# EPICS substitutions: db/ecmcEL37X2_50.substitutions
file ecmcEL37XX-chX.template
{
  pattern { CH_ID, DTYP,             FTVL,  NELM}
          { 1,     asynInt16ArrayIn, SHORT, 50  }
          { 2,     asynInt16ArrayIn, SHORT, 50  }
}
